VAR_GLOBAL
	timer0: TON;
	timer1: TON;
	curTimer: INT := 0;
END_VAR

(* stored: Version 1.1.0.1, ProductVersion 3.1.4022.18
   GVL TIMERS: Id {242fc995-904d-4dd7-8ade-5e22de37db8d} *)
